{ attribute 'Name':='LogMessageBackers-Test' }
{ attribute 'Timeout':='t#5s' }
{ attribute 'Owner':='TestOwner' }
FUNCTION_BLOCK LogMessageBackers_Test EXTENDS FB_TestCaseBase
VAR
	Message : LogMessage;
	expectedMessage : STRING := 'Test';
	expectedSeverity : USINT := 1;
END_VAR

Message.Message	 := expectedMessage;
Message.Severity := expectedSeverity;
AssertMsg(Message.Message = expectedMessage, 'Message getter/setter does NOT work');
AssertMsg(Message.Severity = expectedSeverity, 'Severity getter/setter does NOT work');
Succeeded();

(*Must be implemented if you want to use fastmode*)
METHOD CleanUp : BOOL
CleanUp := TRUE;
END_METHOD

END_FUNCTION_BLOCK

(* stored: Version 1.1.0.1, ProductVersion 3.1.4026.18
   POU LogMessageBackers_Test: Id {fdb3ba85-db9d-4939-a555-4fc38bffee18}, SpecialFunc None
   Method Cleanup: Id {af55f438-5ce1-47fe-a61e-1e93fa6bb622} *)
